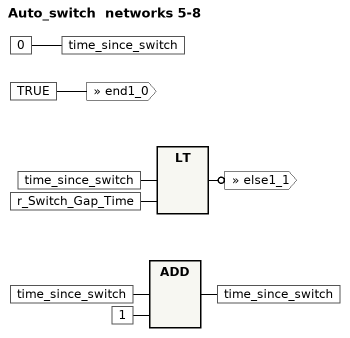
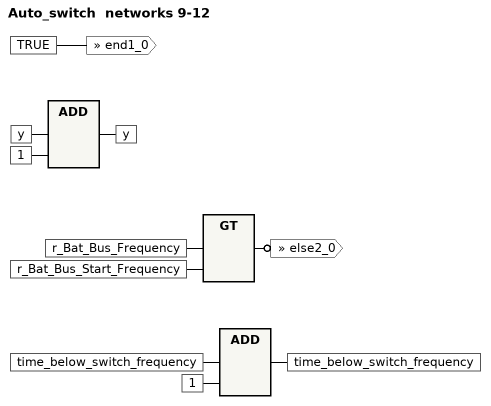
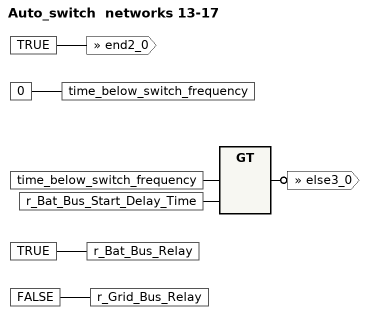
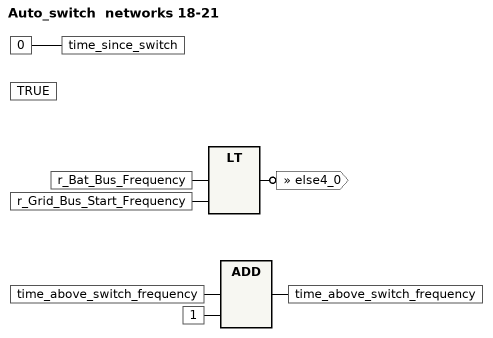
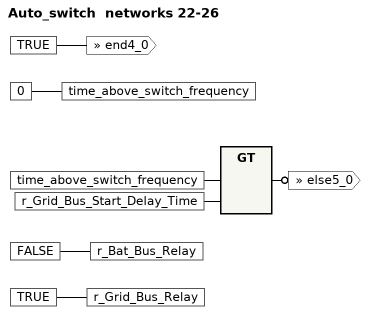
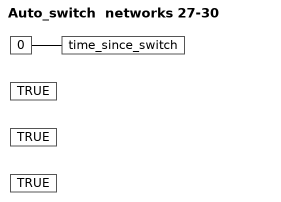
_FBD_ (* Function Block Diagram *)
NETWORK 1 (* this script shuold run every second and / ------ Cases 1 - SAFETY ------ / 1) bat voltage  below 200 	> swtich to gridbus / ------ Cases 2 - NO PENDEL ------ / 2) just switched (wait for r_Switch_Gap_Time) / ------ Cases 3 - LOW FREQUENCY = ENERGY SHORTAGE ------ / 3a) bat frequency below < r_Grid_Bus_Start_Frequency => "reset "to grid counter" / 3b) bat frequency below > r_Grid_Bus_Start_Frequency => "increase "to grid counter" / 3c) "to grid counter" > r_Grid_Bus_Start_Delay_Time => switch of testbus, switch on gridbus relais / ------ Cases 4 - HIGH FREQUENCY = ENERGY SURPLUS ------ / 4a) bat frequency above > r_Bat_Bus_Start_Frequency => "reset "to bat counter" / 4c) "to bat counter" > r_Grid_Bus_Start_Delay_Time => switch of gridbus, switch on testbus relais *)
	ADD(x, 1) => x
NETWORK 2
	NOT LT(r_Bat_Bus_Voltage, 200) => >>else1_0
NETWORK 3 (* case 1 (safety, switching to gridbus) *)
	FALSE => r_Bat_Bus_Relay
NETWORK 4
	TRUE => r_Grid_Bus_Relay
NETWORK 5
	0 => time_since_switch
NETWORK 6
	TRUE => >>end1_0
NETWORK 7 else1_0::
	NOT LT(time_since_switch, r_Switch_Gap_Time) => >>else1_1
NETWORK 8 (* case 2 (already switched recently) *)
	ADD(time_since_switch, 1) => time_since_switch
NETWORK 9
	TRUE => >>end1_0
NETWORK 10 else1_1::
	ADD(y, 1) => y
NETWORK 11 (* CASE 3 / 3a+b *)
	NOT GT(r_Bat_Bus_Frequency, r_Bat_Bus_Start_Frequency) => >>else2_0
NETWORK 12
	ADD(time_below_switch_frequency, 1) => time_below_switch_frequency
NETWORK 13
	TRUE => >>end2_0
NETWORK 14 else2_0::
	0 => time_below_switch_frequency
NETWORK 15 end2_0:: (* 3C time_below_switch_frequency passed >> switching *)
	NOT GT(time_below_switch_frequency, r_Bat_Bus_Start_Delay_Time) => >>else3_0
NETWORK 16
	TRUE => r_Bat_Bus_Relay
NETWORK 17
	FALSE => r_Grid_Bus_Relay
NETWORK 18
	0 => time_since_switch
NETWORK 19 end3_0::
	TRUE
NETWORK 20 else3_0:: (* CASE 4 / 4a+b *)
	NOT LT(r_Bat_Bus_Frequency, r_Grid_Bus_Start_Frequency) => >>else4_0
NETWORK 21
	ADD(time_above_switch_frequency, 1) => time_above_switch_frequency
NETWORK 22
	TRUE => >>end4_0
NETWORK 23 else4_0::
	0 => time_above_switch_frequency
NETWORK 24 end4_0:: (* 4C time_above_switch_frequency passed >> switching *)
	NOT GT(time_above_switch_frequency, r_Grid_Bus_Start_Delay_Time) => >>else5_0
NETWORK 25
	FALSE => r_Bat_Bus_Relay
NETWORK 26
	TRUE => r_Grid_Bus_Relay
NETWORK 27
	0 => time_since_switch
NETWORK 28 end5_0::
	TRUE
NETWORK 29 end1_0::
	TRUE
NETWORK 30 else5_0::
	TRUE
_END_FBD_
END_PROGRAM

(* POU 04. Frequency based Bus Select/Auto_switch_delay, ST *)
PROGRAM Auto_switch_delay
(* ____________________________  USED GLOBAL VARIABLES  ___________________________

VAR_INPUT

	CHP_new_state_grid_bus							:	BOOL; (* request based on frequency *)
	CHP_new_state_battery_bus						:	BOOL; (* request based on frequency *)

	CHP_relay_state_battery_bus   							AT %IX134.1  : BOOL;  (* INVERTED INPUTS *)
	CHP_relay_state_grid_bus   								AT %IX134.2  : BOOL;  (* INVERTED INPUTS *)
	
	CHP_control_internal_contacter_switch_state

END_VAR

VAR_OUTPUT

	Group1_3F_Auto_relay_control_battery_bus							:	BOOL; (* request based on frequency, has delayed switching!! *)
	Group1_3F_Auto_relay_control_battery_bus							:	BOOL; (* request based on frequency, has delayed switching!! *)

END_VAR
*)

VAR
	y: BOOL :=FALSE;
	z: INT;
END_VAR
(* CHP handler uses frequency based switching input to control real CHP swithcing when auto input is high *)
(* CHP handler delays switching, such that the CHP can depower and disconnect before switch *)
(* CHP handler delays on-switching, making sure the CHP is disconnected. *)
(* CHP handler delays on-switching, making sure the CHP will connect to the right bus (in the right mode). *)

(* ____________________________  AUTO SWITCH CONTROL  ___________________________ *)
IF Group1_3F_Selector_auto_bus_select = TRUE THEN
	z := z + 1;
	(*check if wanted state to CHP signal is right, change when required *)
	IF CHP_new_state_grid_bus =TRUE THEN
		CHP_control_Offgrid_request :=FALSE;
		z :=0;
		y := FALSE;
	ELSE
		IF CHP_new_state_battery_bus = TRUE THEN
		CHP_control_Offgrid_request :=TRUE;
		z := 100;
		y := TRUE;
		END_IF;
	END_IF;

	(* perform switch between busses when CHP has disconnceted *)
	IF CHP_control_internal_contacter_switch_state = FALSE THEN

		(* Close bat relais when grid relais is open en bat request is still true*)
		IF CHP_new_state_battery_bus =TRUE  THEN

			IF CHP_relay_state_grid_bus = TRUE THEN (* INVERTED INPUTS *)
				Group1_3F_Auto_relay_control_battery_bus := TRUE;
			END_IF;
			Group1_3F_Auto_relay_control_grid_bus := FALSE; (* Disconnect GRID SCWICH*)
		END_IF;

		(* Close grid relais when bat relais is open en grid request is still true*)
		IF CHP_new_state_grid_bus =TRUE  THEN

			IF CHP_relay_state_battery_bus = TRUE THEN (* INVERTED INPUTS *)
				Group1_3F_Auto_relay_control_grid_bus := TRUE;
			END_IF;
			Group1_3F_Auto_relay_control_battery_bus := FALSE; (* Disconnect *)
		END_IF;
	END_IF;


(* ____________________________  MANUAL CONTROL  ___________________________ *)
ELSE
	z := 200;
	(* check if batbus relais is closed, if so, request offgrid (via wanted state *)
	IF Group1_3F_relay_state_battery_bus = TRUE THEN
		CHP_control_Offgrid_request :=TRUE;
	ELSE (* IF Group1_3F_relay_state_grid_bus THEN *)
		CHP_control_Offgrid_request :=FALSE;
	END_IF;

	Group1_3F_Auto_relay_control_grid_bus := FALSE; (* Disconnect GRID SCWICH*)
	Group1_3F_Auto_relay_control_battery_bus := FALSE; (* Disconnect *)
END_IF;
END_PROGRAM

(* POU 02. Batterybus Frequency to Analog Out/EV_Controller, FBD *)
PROGRAM EV_Controller
VAR
	RAMP_REAL: RAMP_REAL;
	Frequency_to_Analog_Out: Frequency_to_Analog_Out;
	EV_control_control_signal2: INT;
	RAMP_WORD4: RAMP_INT;
END_VAR
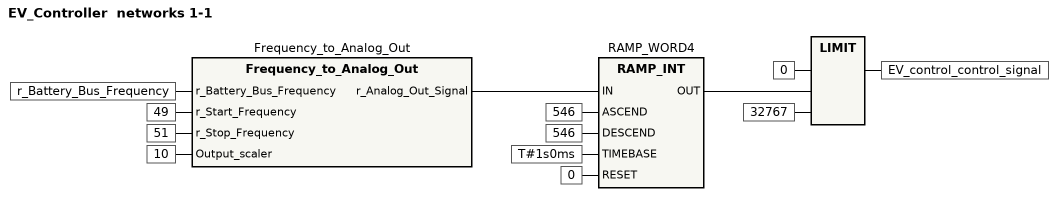
_FBD_ (* Function Block Diagram *)
NETWORK 1
	LIMIT(0, RAMP_WORD4:RAMP_INT(IN: Frequency_to_Analog_Out:Frequency_to_Analog_Out(r_Battery_Bus_Frequency: r_Battery_Bus_Frequency, r_Start_Frequency: 49, r_Stop_Frequency: 51, Output_scaler: 10), ASCEND: 546, DESCEND: 546, TIMEBASE: T#1s0ms, RESET: 0), 32767) => EV_control_control_signal
_END_FBD_
(* the same logic as Structured Text *)
(* Network 1 *)
Frequency_to_Analog_Out(r_Battery_Bus_Frequency := r_Battery_Bus_Frequency, r_Start_Frequency := 49, r_Stop_Frequency := 51, Output_scaler := 10);
RAMP_WORD4(IN := Frequency_to_Analog_Out.r_Analog_Out_Signal, ASCEND := 546, DESCEND := 546, TIMEBASE := T#1s0ms, RESET := 0);
EV_control_control_signal := LIMIT(0, RAMP_WORD4.OUT, 32767);
END_PROGRAM

(* POU 04. Frequency based Bus Select/GroupTest, FBD *)
PROGRAM GroupTest
VAR

	request_grid: BOOL;
	request_testbus: BOOL;
	Delayer: Auto_delayer;
	Switch: Auto_switch_new;
END_VAR
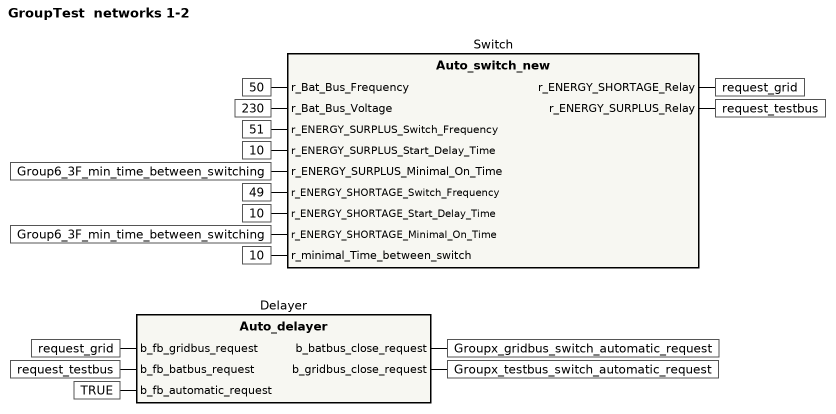
_FBD_ (* Function Block Diagram *)
NETWORK 1
	Switch:Auto_switch_new(r_Bat_Bus_Frequency: 50, r_Bat_Bus_Voltage: 230, r_ENERGY_SURPLUS_Switch_Frequency: 51, r_ENERGY_SURPLUS_Start_Delay_Time: 10, r_ENERGY_SURPLUS_Minimal_On_Time: Group6_3F_min_time_between_switching, r_ENERGY_SHORTAGE_Switch_Frequency: 49, r_ENERGY_SHORTAGE_Start_Delay_Time: 10, r_ENERGY_SHORTAGE_Minimal_On_Time: Group6_3F_min_time_between_switching, r_minimal_Time_between_switch: 10, r_ENERGY_SURPLUS_Relay => request_testbus) => request_grid
NETWORK 2
	Delayer:Auto_delayer(b_fb_gridbus_request: request_grid, b_fb_batbus_request: request_testbus, b_fb_automatic_request: TRUE, b_gridbus_close_request => Groupx_testbus_switch_automatic_request) => Groupx_gridbus_switch_automatic_request
_END_FBD_
(* the same logic as Structured Text *)
(* Network 1 *)
Switch(r_Bat_Bus_Frequency := 50, r_Bat_Bus_Voltage := 230, r_ENERGY_SURPLUS_Switch_Frequency := 51, r_ENERGY_SURPLUS_Start_Delay_Time := 10, r_ENERGY_SURPLUS_Minimal_On_Time := Group6_3F_min_time_between_switching, r_ENERGY_SHORTAGE_Switch_Frequency := 49, r_ENERGY_SHORTAGE_Start_Delay_Time := 10, r_ENERGY_SHORTAGE_Minimal_On_Time := Group6_3F_min_time_between_switching, r_minimal_Time_between_switch := 10);
request_testbus := Switch.r_ENERGY_SURPLUS_Relay;
request_grid := Switch.r_ENERGY_SHORTAGE_Relay;
(* Network 2 *)
Delayer(b_fb_gridbus_request := request_grid, b_fb_batbus_request := request_testbus, b_fb_automatic_request := TRUE);
Groupx_testbus_switch_automatic_request := Delayer.b_gridbus_close_request;
Groupx_gridbus_switch_automatic_request := Delayer.b_batbus_close_request;
END_PROGRAM

(* POU 04. Frequency based Bus Select/init, ST *)
PROGRAM init
VAR

END_VAR
(* frequency based switching is deactivated BY default AND can be activated via modbus *)
IF initialized = FALSE THEN
arSystemState[246] :=Group_control_Frequencybased_bus_selecting_state;  (* default is off *)
arSystemState[247] :=Group_control_min_time_above_switch_frequency;
arSystemState[248] :=Group_control_min_time_below_switch_frequency;
arSystemState[249] :=Group1_3F_Switch_frequency_to_batterybus;
arSystemState[250] :=Group1_3F_Switch_frequency_to_gridbus;
arSystemState[251] :=Group1_3F_min_time_between_switching;
arSystemState[252] :=Group2_3F_Switch_frequency_to_batterybus;
arSystemState[253] :=Group2_3F_Switch_frequency_to_gridbus;
arSystemState[254] :=Group2_3F_min_time_between_switching;
arSystemState[253] :=Group3_3F_Switch_frequency_to_batterybus;
arSystemState[254] :=Group3_3F_Switch_frequency_to_gridbus;
arSystemState[255] :=Group3_3F_min_time_between_switching;
arSystemState[256] :=Group4_3F_Switch_frequency_to_batterybus;
arSystemState[255] :=Group4_3F_Switch_frequency_to_gridbus;
arSystemState[256] :=Group4_3F_min_time_between_switching;
arSystemState[257] :=Group5_3F_Switch_frequency_to_batterybus;
arSystemState[258] :=Group5_3F_Switch_frequency_to_gridbus;
arSystemState[257] :=Group5_3F_min_time_between_switching;
arSystemState[258] :=Group6_3F_Switch_frequency_to_batterybus;
arSystemState[259] :=Group6_3F_Switch_frequency_to_gridbus;
arSystemState[260] :=Group6_3F_min_time_between_switching;
arSystemState[259] :=Group7_3F_Switch_frequency_to_batterybus;
arSystemState[260] :=Group7_3F_Switch_frequency_to_gridbus;
arSystemState[261] :=Group7_3F_min_time_between_switching;
arSystemState[262] :=Group8_3F_Switch_frequency_to_batterybus;
arSystemState[261] :=Group8_3F_Switch_frequency_to_gridbus;
arSystemState[262] :=Group8_3F_min_time_between_switching;
arSystemState[263] :=Group9_3F_Switch_frequency_to_batterybus;
arSystemState[264] :=Group9_3F_Switch_frequency_to_gridbus;
arSystemState[263] :=Group9_3F_min_time_between_switching;
initialized := TRUE;
END_IF;
END_PROGRAM

(* POU Configuration/MODBUS_CONFIGURATION, ST *)
PROGRAM MODBUS_CONFIGURATION
VAR                                
END_VAR                            
(*                                 
   <?xml version="1.0" encoding="UTF-16" standalone="yes"?>
<network xml_structure_version="1" xml_feature_version="1">
	<generator_settings minRTUTaskCycleTimeMs="100" minEthaskCycleTimeMs="5" ethSlaveMultiplier="0.1" rtuInterfaceMultiplier="0.1" taskGeneration="false"/>
	<master_interface type="eth" name="" expanded="true">
		<mb_slave comment="" name="Janitza_UMG5090" expanded="true" type="generic">
			<mb_connection type="eth" transport="UDP" port="502" ip="192.168.1.2" unitid="1" request_delay_ms="0" response_timeout_ms="20"/>
			<generic_vars comment="" expanded="true">
				<generic_var data_type="REAL">
					<generic_params name="PactiveL1" comment="" expanded="false" mb_iotype="unused" mb_access="ro" var_byteorder="B3B4B1B2"/>
					<mb_address explicitAccess="false" FCRead="3" FCWrite="0" ReadMBAddress="2069" WriteMBAddress="0" ReadBitOffset="0" WriteBitOffset="0"/>
				</generic_var>
				<generic_var data_type="REAL">
					<generic_params name="PactiveL2" comment="" expanded="true" mb_iotype="unused" mb_access="ro" var_byteorder="B3B4B1B2"/>
					<mb_address explicitAccess="false" FCRead="3" FCWrite="0" ReadMBAddress="2071" WriteMBAddress="0" ReadBitOffset="0" WriteBitOffset="0"/>
				</generic_var>
				<generic_var data_type="REAL">
					<generic_params name="PactiveL3" comment="" expanded="true" mb_iotype="unused" mb_access="ro" var_byteorder="B3B4B1B2"/>
					<mb_address explicitAccess="false" FCRead="3" FCWrite="0" ReadMBAddress="2073" WriteMBAddress="0" ReadBitOffset="0" WriteBitOffset="0"/>
				</generic_var>
				<generic_var data_type="REAL">
					<generic_params name="PreactiveL1" comment="" expanded="false" mb_iotype="unused" mb_access="ro" var_byteorder="B3B4B1B2"/>
					<mb_address explicitAccess="false" FCRead="3" FCWrite="0" ReadMBAddress="2077" WriteMBAddress="0" ReadBitOffset="0" WriteBitOffset="0"/>
				</generic_var>
				<generic_var data_type="REAL">
					<generic_params name="PreactiveL2" comment="" expanded="true" mb_iotype="unused" mb_access="ro" var_byteorder="B3B4B1B2"/>
					<mb_address explicitAccess="false" FCRead="3" FCWrite="0" ReadMBAddress="2079" WriteMBAddress="0" ReadBitOffset="0" WriteBitOffset="0"/>
				</generic_var>
				<generic_var data_type="REAL">
					<generic_params name="PreactiveL3" comment="" expanded="true" mb_iotype="unused" mb_access="ro" var_byteorder="B3B4B1B2"/>
					<mb_address explicitAccess="false" FCRead="3" FCWrite="0" ReadMBAddress="2081" WriteMBAddress="0" ReadBitOffset="0" WriteBitOffset="0"/>
				</generic_var>
				<generic_var data_type="REAL">
					<generic_params name="VoltageL1" comment="" expanded="true" mb_iotype="unused" mb_access="ro" var_byteorder="B3B4B1B2"/>
					<mb_address explicitAccess="false" FCRead="3" FCWrite="0" ReadMBAddress="2053" WriteMBAddress="0" ReadBitOffset="0" WriteBitOffset="0"/>
				</generic_var>
				<generic_var data_type="REAL">
					<generic_params name="VoltageL2" comment="" expanded="false" mb_iotype="unused" mb_access="ro" var_byteorder="B3B4B1B2"/>
					<mb_address explicitAccess="false" FCRead="3" FCWrite="0" ReadMBAddress="2055" WriteMBAddress="0" ReadBitOffset="0" WriteBitOffset="0"/>
				</generic_var>
				<generic_var data_type="REAL">
					<generic_params name="VoltageL3" comment="" expanded="false" mb_iotype="unused" mb_access="ro" var_byteorder="B3B4B1B2"/>
					<mb_address explicitAccess="false" FCRead="3" FCWrite="0" ReadMBAddress="2057" WriteMBAddress="0" ReadBitOffset="0" WriteBitOffset="0"/>
				</generic_var>
				<generic_var data_type="REAL">
					<generic_params name="VoltageL4" comment="" expanded="false" mb_iotype="unused" mb_access="ro" var_byteorder="B3B4B1B2"/>
					<mb_address explicitAccess="false" FCRead="3" FCWrite="0" ReadMBAddress="2059" WriteMBAddress="0" ReadBitOffset="0" WriteBitOffset="0"/>
				</generic_var>
				<generic_var data_type="REAL">
					<generic_params name="PhaseCurrentL1" comment="" expanded="true" mb_iotype="unused" mb_access="ro" var_byteorder="B3B4B1B2"/>
					<mb_address explicitAccess="false" FCRead="3" FCWrite="0" ReadMBAddress="2061" WriteMBAddress="0" ReadBitOffset="0" WriteBitOffset="0"/>
				</generic_var>
				<generic_var data_type="REAL">
					<generic_params name="PhaseCurrentL2" comment="" expanded="true" mb_iotype="unused" mb_access="ro" var_byteorder="B3B4B1B2"/>
					<mb_address explicitAccess="false" FCRead="3" FCWrite="0" ReadMBAddress="2063" WriteMBAddress="0" ReadBitOffset="0" WriteBitOffset="0"/>
				</generic_var>
				<generic_var data_type="REAL">
					<generic_params name="PhaseCurrentL3" comment="" expanded="true" mb_iotype="unused" mb_access="ro" var_byteorder="B3B4B1B2"/>
					<mb_address explicitAccess="false" FCRead="3" FCWrite="0" ReadMBAddress="2065" WriteMBAddress="0" ReadBitOffset="0" WriteBitOffset="0"/>
				</generic_var>
				<generic_var data_type="REAL">
					<generic_params name="PhaseCurrentLN" comment="" expanded="true" mb_iotype="unused" mb_access="ro" var_byteorder="B3B4B1B2"/>
					<mb_address explicitAccess="false" FCRead="3" FCWrite="0" ReadMBAddress="2067" WriteMBAddress="0" ReadBitOffset="0" WriteBitOffset="0"/>
				</generic_var>
				<generic_var data_type="REAL">
					<generic_params name="FieldRotation" comment="" expanded="true" mb_iotype="unused" mb_access="ro" var_byteorder="B3B4B1B2"/>
					<mb_address explicitAccess="false" FCRead="3" FCWrite="0" ReadMBAddress="2185" WriteMBAddress="0" ReadBitOffset="0" WriteBitOffset="0"/>
				</generic_var>
				<generic_var data_type="REAL">
					<generic_params name="CosPihL1" comment="" expanded="true" mb_iotype="unused" mb_access="ro" var_byteorder="B3B4B1B2"/>
					<mb_address explicitAccess="false" FCRead="3" FCWrite="0" ReadMBAddress="2159" WriteMBAddress="0" ReadBitOffset="0" WriteBitOffset="0"/>
				</generic_var>
				<generic_var data_type="REAL">
					<generic_params name="CosPihL2" comment="" expanded="true" mb_iotype="unused" mb_access="ro" var_byteorder="B3B4B1B2"/>
					<mb_address explicitAccess="false" FCRead="3" FCWrite="0" ReadMBAddress="2161" WriteMBAddress="0" ReadBitOffset="0" WriteBitOffset="0"/>
				</generic_var>
				<generic_var data_type="REAL">
					<generic_params name="CosPihL3" comment="" expanded="true" mb_iotype="unused" mb_access="ro" var_byteorder="B3B4B1B2"/>
					<mb_address explicitAccess="false" FCRead="3" FCWrite="0" ReadMBAddress="2163" WriteMBAddress="0" ReadBitOffset="0" WriteBitOffset="0"/>
				</generic_var>
				<generic_var data_type="REAL">
					<generic_params name="Frequency" comment="" expanded="true" mb_iotype="unused" mb_access="ro" var_byteorder="B3B4B1B2"/>
					<mb_address explicitAccess="false" FCRead="3" FCWrite="0" ReadMBAddress="2175" WriteMBAddress="0" ReadBitOffset="0" WriteBitOffset="0"/>
				</generic_var>
				<generic_var data_type="REAL">
					<generic_params name="PactivetTot" comment="" expanded="false" mb_iotype="unused" mb_access="ro" var_byteorder="B3B4B1B2"/>
					<mb_address explicitAccess="false" FCRead="3" FCWrite="0" ReadMBAddress="2105" WriteMBAddress="0" ReadBitOffset="0" WriteBitOffset="0"/>
				</generic_var>
				<generic_var data_type="REAL">
					<generic_params name="PactivetTotL4" comment="" expanded="false" mb_iotype="unused" mb_access="ro" var_byteorder="B3B4B1B2"/>
					<mb_address explicitAccess="false" FCRead="3" FCWrite="0" ReadMBAddress="2113" WriteMBAddress="0" ReadBitOffset="0" WriteBitOffset="0"/>
				</generic_var>
			</generic_vars>
		</mb_slave>
	</master_interface>
</network>
                              
*)                                 
;                                  
END_PROGRAM

(* POU 02. Batterybus Frequency to Analog Out/other_control_signal, FBD *)
PROGRAM other_control_signal
VAR
	RAMP_REAL: RAMP_REAL;
	Frequency_to_Analog_Out: Frequency_to_Analog_Out;
END_VAR
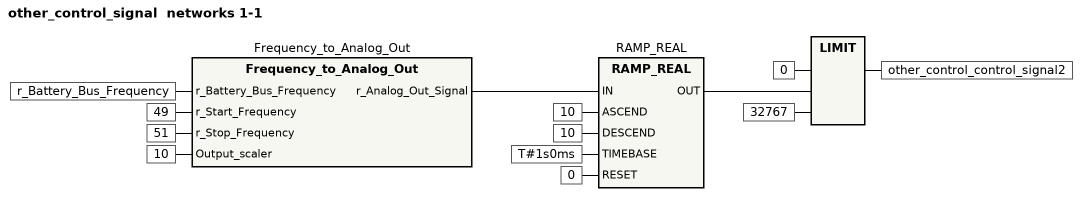
_FBD_ (* Function Block Diagram *)
NETWORK 1
	LIMIT(0, RAMP_REAL:RAMP_REAL(IN: Frequency_to_Analog_Out:Frequency_to_Analog_Out(r_Battery_Bus_Frequency: r_Battery_Bus_Frequency, r_Start_Frequency: 49, r_Stop_Frequency: 51, Output_scaler: 10), ASCEND: 10, DESCEND: 10, TIMEBASE: T#1s0ms, RESET: 0), 32767) => other_control_control_signal2
_END_FBD_
(* the same logic as Structured Text *)
(* Network 1 *)
Frequency_to_Analog_Out(r_Battery_Bus_Frequency := r_Battery_Bus_Frequency, r_Start_Frequency := 49, r_Stop_Frequency := 51, Output_scaler := 10);
RAMP_REAL(IN := Frequency_to_Analog_Out.r_Analog_Out_Signal, ASCEND := 10, DESCEND := 10, TIMEBASE := T#1s0ms, RESET := 0);
other_control_control_signal2 := LIMIT(0, RAMP_REAL.OUT, 32767);
END_PROGRAM

(* POU TheBattery/SOC_real_to_Voltage_Out, ST *)
PROGRAM SOC_real_to_Voltage_Out
VAR

END_VAR
other_control_control_signal := REAL_TO_WORD(6553.6*TheBattery_SOC_real/10);
END_PROGRAM

(* POU 03. Synchroniser Switch control/SynchronizerModbusStateHandler_PRG, ST *)
PROGRAM SynchronizerModbusStateHandler_PRG
VAR

END_VAR
(*___OLD___
IF r_modbus_Synchroniser_state < 1 THEN
		r_modbus_Synchroniser_Denied_Request := TRUE;
		r_modbus_Synchroniser_Close_Request := FALSE;
ELSE
	IF r_modbus_Synchroniser_state > 1.99 THEN
		r_modbus_Synchroniser_Denied_Request := FALSE;
		r_modbus_Synchroniser_Close_Request := TRUE;
	ELSE
		r_modbus_Synchroniser_Denied_Request := FALSE;
		r_modbus_Synchroniser_Close_Request := FALSE;
	END_IF
END_IF
*)
END_PROGRAM

(* POU 04. Frequency based Bus Select/Test, ST *)
PROGRAM Test
VAR

	Test :fbSwitchRelaysBatOrGridBus;
	a: REAL;
	frequencybased_bus_selecting_state: BOOL;
END_VAR
	frequencybased_bus_selecting_state : = arSystemState[999]; (* frequency based switching is deactivated by default and can be activated via modbus *)


Test(
	r_Off_Grid_Bus_Frequency:= r_Battery_Bus_Frequency ,
	r_Off_Grid_Bus_Voltage:= 250,
	r_On_Grid_Start_Frequency:= 49,
	r_On_Grid_Start_Delay_Time:= 2000,
	r_On_Grid_Minimal_On_Time:= 2000 ,
	r_Off_Grid_Start_Frequency:= 51,
	r_Off_Grid_Start_Delay_Time:= 2000,
	r_Switch_Gap_Time:= 2000,
	r_Off_Grid_Minimal_On_Time:= 2000);

(*
	Group1_Switch_frequency_to_batterybus						:  read from mobus;
	Group1_Switch_frequency_to_gridbus							:  REAL 	:= 48;
	Group1_min_time_above_switch frequency						:  INT 		: = 10000; (*ms*)
	Group1_min_time_below_switch frequency						:  INT 		: = 10000; (*ms*)
	Group1_min_time_between_switching							:  INT 		: = 10000; (*ms*)
*)
END_PROGRAM

(* POU 04. Frequency based Bus Select/fbSwitchRelaysBatOrGridBus, SFC *)
FUNCTION_BLOCK fbSwitchRelaysBatOrGridBus
VAR_INPUT

	r_Bat_Bus_Frequency						:	REAL;
	r_Bat_Bus_Voltage							:	REAL;
	r_Grid_Bus_Start_Frequency					:	REAL;
	r_Grid_Bus_Start_Delay_Time				:	REAL;
	r_Grid_Bus_Minimal_On_Time				:	REAL;
	r_Bat_Bus_Start_Frequency					:	REAL;
	r_Bat_Bus_Start_Delay_Time				:	REAL;
	r_Bat_Bus_Minimal_On_Time				:	REAL;
	r_Switch_Gap_Time							: 	REAL;		(* Time between on and off grid relay switching (dead bus gap) *)

END_VAR
VAR_OUTPUT

	r_Grid_Bus_Relay								:	BOOL := TRUE;
	r_Bat_Bus_Relay									:	BOOL;

END_VAR
VAR
	r_Bat_Bus_Min_Voltage 							: 	REAL :=200;
	r_Checked_Grid_Bus_Start_Frequency			:	REAL;
	r_Checked_Bat_Bus_Start_Frequency			:	REAL;

	t_Grid_Bus_Start_Delay_Timer					:	TON;
	t_Bat_Bus_Start_Delay_Timer					:	TON;

END_VAR
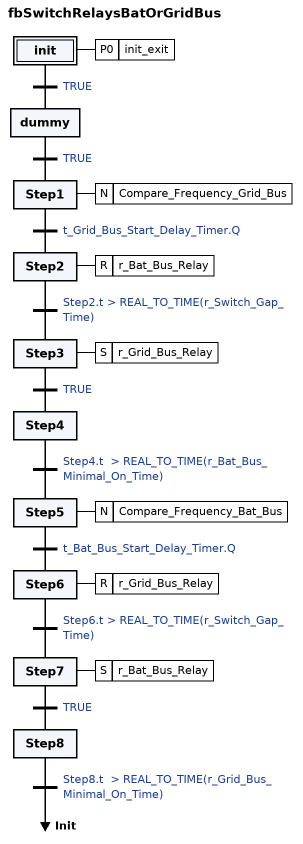
INITIAL_STEP init:
	init_exit(P0);
END_STEP
TRANSITION FROM init TO dummy := TRUE;
END_TRANSITION
STEP dummy:
END_STEP
TRANSITION FROM dummy TO Step1 := TRUE;
END_TRANSITION
STEP Step1:
	Compare_Frequency_Grid_Bus(N);
END_STEP
TRANSITION FROM Step1 TO Step2 := t_Grid_Bus_Start_Delay_Timer.Q;
END_TRANSITION
STEP Step2:
	r_Bat_Bus_Relay(R);
END_STEP
TRANSITION FROM Step2 TO Step3 := Step2.t > REAL_TO_TIME(r_Switch_Gap_Time);
END_TRANSITION
STEP Step3:
	r_Grid_Bus_Relay(S);
END_STEP
TRANSITION FROM Step3 TO Step4 := TRUE;
END_TRANSITION
STEP Step4:
END_STEP
TRANSITION FROM Step4 TO Step5 := Step4.t  > REAL_TO_TIME(r_Bat_Bus_Minimal_On_Time);
END_TRANSITION
STEP Step5:
	Compare_Frequency_Bat_Bus(N);
END_STEP
TRANSITION FROM Step5 TO Step6 := t_Bat_Bus_Start_Delay_Timer.Q;
END_TRANSITION
STEP Step6:
	r_Grid_Bus_Relay(R);
END_STEP
TRANSITION FROM Step6 TO Step7 := Step6.t > REAL_TO_TIME(r_Switch_Gap_Time);
END_TRANSITION
STEP Step7:
	r_Bat_Bus_Relay(S);
END_STEP
TRANSITION FROM Step7 TO Step8 := TRUE;
END_TRANSITION
STEP Step8:
END_STEP
TRANSITION FROM Step8 TO Init := Step8.t  > REAL_TO_TIME(r_Grid_Bus_Minimal_On_Time);
END_TRANSITION

ACTION init_exit:
(* Bat_Bus start frequency should by higher than grid bus start frequency to prevent pendel behaviour of states *)

IF r_Bat_Bus_Start_Frequency > r_Grid_Bus_Start_Frequency THEN

	r_Checked_Bat_Bus_Start_Frequency := r_Bat_Bus_Start_Frequency;
	r_Checked_Grid_Bus_Start_Frequency := r_Grid_Bus_Start_Frequency;

ELSE

	r_Checked_Bat_Bus_Start_Frequency := r_Bat_Bus_Start_Frequency;
	r_Checked_Grid_Bus_Start_Frequency := r_Bat_Bus_Start_Frequency;

END_IF
END_ACTION
END_FUNCTION_BLOCK
ACTION Compare_Frequencies:
(* Bat_Bus start frequency should by higher than grid bus start frequency to prevent pendel behaviour of states *)

IF r_Bat_Bus_Start_Frequency > r_Grid_Bus_Start_Frequency THEN

	r_Checked_Bat_Bus_Start_Frequency := r_Bat_Bus_Start_Frequency;
	r_Checked_Grid_Bus_Start_Frequency := r_Grid_Bus_Start_Frequency;

ELSE

	r_Checked_Bat_Bus_Start_Frequency := r_Bat_Bus_Start_Frequency;
	r_Checked_Grid_Bus_Start_Frequency := r_Bat_Bus_Start_Frequency;

END_IF
END_ACTION
ACTION Compare_Frequency_Bat_Bus:
t_Bat_Bus_Start_Delay_Timer(
	IN:= r_Bat_Bus_Frequency > r_Checked_Bat_Bus_Start_Frequency AND r_Bat_Bus_Voltage > r_Bat_Bus_Min_Voltage,
	PT:= REAL_TO_TIME(r_Bat_Bus_Start_Delay_Time));
END_ACTION
ACTION Compare_Frequency_Grid_Bus:
t_Grid_Bus_Start_Delay_Timer(
	IN:= r_Bat_Bus_Frequency < r_Checked_Grid_Bus_Start_Frequency,
	PT:= REAL_TO_TIME(r_Grid_Bus_Start_Delay_Time));
END_ACTION
ACTION Compare_Frequency_Grid_Bus_old:
t_Grid_Bus_Start_Delay_Timer(
	IN:= r_Bat_Bus_Frequency < r_Checked_Grid_Bus_Start_Frequency,
	PT:= REAL_TO_TIME(r_Grid_Bus_Start_Delay_Time));
END_ACTION
ACTION Compare_Frequency_Grid_Bus_olds:
t_Grid_Bus_Start_Delay_Timer(
	IN:= r_Bat_Bus_Frequency < r_Checked_Grid_Bus_Start_Frequency,
	PT:= REAL_TO_TIME(r_Grid_Bus_Start_Delay_Time));
END_ACTION

(* POU 04. Frequency based Bus Select/test_switch, LD *)
PROGRAM test_switch
VAR
	test: CHP_Switch_Handler;
END_VAR
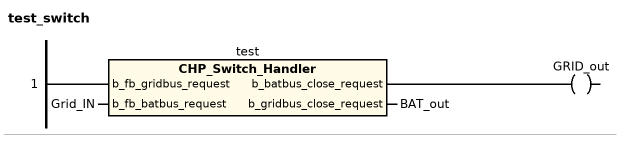
_LD_ (* Ladder Diagram *)
NETWORK 1
	test:CHP_Switch_Handler(b_fb_gridbus_request: *, b_fb_batbus_request: Grid_IN, b_gridbus_close_request => BAT_out) --- (GRID_out)
_END_LD_
(* the same logic as Structured Text *)
(* Network 1 *)
test(b_fb_gridbus_request := TRUE, b_fb_batbus_request := Grid_IN);
BAT_out := test.b_gridbus_close_request;
GRID_out := test.b_batbus_close_request;
END_PROGRAM

(* POU 04. Frequency based Bus Select/CHP_Switch_Handler, ST *)
FUNCTION_BLOCK CHP_Switch_Handler

VAR_INPUT

	b_fb_gridbus_request							:	BOOL; (* request based on frequency, has delayed switching!! *)
	b_fb_batbus_request								:	BOOL; (* request based on frequency, has delayed switching!! *)

END_VAR

VAR_OUTPUT

	b_batbus_close_request							:	BOOL; (* request based on frequency, has delayed switching!! *)
	b_gridbus_close_request							:	BOOL; (* request based on frequency, has delayed switching!! *)

END_VAR

VAR
(* ____________________________  USED GLOBAL VARIABLES  ___________________________ *)
(*
	(* INPUTS *)
	CHP_control_internal_contacter_switch_state  			AT %IX121.15 : BOOL;
	Group1_3F_Selector_auto_bus_select    				AT %IX121.2 : BOOL;
	Group1_3F_relay_state_battery_bus   					AT %IX120.1  : BOOL;
	Group1_3F_relay_state_grid_bus   						AT %IX120.0  : BOOL;

	(* OUTPUTS *)
	Group1_3F_Auto_relay_control_battery_bus   			AT %QX128.1  : BOOL;
	Group1_3F_Auto_relay_control_grid_bus   				AT %QX128.0  : BOOL;
	CHP_control_Offgrid_request    							AT %QX129.4  : BOOL;
*)
	y: BOOL :=FALSE;
	z: INT;
END_VAR
(* CHP handler uses frequency based switching input to control real CHP swithcing when auto input is high *)
(* CHP handler delays switching, such that the CHP can depower and disconnect before switch *)
(* CHP handler delays on-switching, making sure the CHP is disconnected. *)
(* CHP handler delays on-switching, making sure the CHP will connect to the right bus (in the right mode). *)

(* ____________________________  AUTO SWITCH CONTROL  ___________________________ *)
IF Group1_3F_Selector_auto_bus_select = TRUE THEN
	z := z + 1;
	(*check if wanted state to CHP signal is right, change when required *)
	IF b_fb_gridbus_request =TRUE THEN
		CHP_control_Offgrid_request :=FALSE;
		z :=0;
		y := FALSE;
	ELSE
		IF b_fb_batbus_request = TRUE THEN
		CHP_control_Offgrid_request :=TRUE;
		z := 100;
		y := TRUE;
		END_IF;
	END_IF;

	(* perform switch between busses when CHP has disconnceted *)
	IF CHP_control_internal_contacter_switch_state = FALSE THEN

		(* Close bat relais when grid relais is open en bat request is still true*)
		IF b_fb_batbus_request =TRUE  THEN
			b_gridbus_close_request := FALSE; (* Disconnect GRID SCWICH*)
			IF Group1_3F_relay_state_grid_bus = FALSE THEN
				b_batbus_close_request := TRUE;
			END_IF;
		END_IF;

		(* Close grid relais when bat relais is open en grid request is still true*)
		IF b_fb_gridbus_request =TRUE  THEN
			b_batbus_close_request := FALSE; (* Disconnect *)
			IF Group1_3F_relay_state_battery_bus = FALSE THEN
				b_gridbus_close_request := TRUE;
			END_IF;
		END_IF;
	END_IF;


(* ____________________________  MANUAL CONTROL  ___________________________ *)
ELSE
	z := 200;
	(* check if batbus relais is closed, if so, request offgrid (via wanted state *)
	IF Group1_3F_relay_state_battery_bus = TRUE THEN
		CHP_control_Offgrid_request :=TRUE;
	ELSE (* IF Group1_3F_relay_state_grid_bus THEN *)
		CHP_control_Offgrid_request :=FALSE;
	END_IF;
END_IF;
END_FUNCTION_BLOCK

(* POU 08. SD CARD logging/WRITE_CSV/WRITE_DATA, FBD *)
PROGRAM WRITE_DATA
VAR
	FB1				: FbDatalogger;
	xGo				: BOOL		:= TRUE;
	xTrigger			: BOOL;
	Channels			: ARRAY [1.. 80] OF typUserInput;
	Settings			: typConfigDatalogger;
	bDType			: BYTE := 1;
	xFirstCycle			: BOOL := TRUE;
	i: INT;

END_VAR
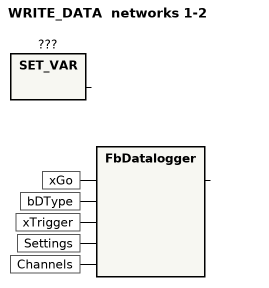
_FBD_ (* Function Block Diagram *)
NETWORK 1
	???:SET_VAR()
NETWORK 2
	FbDatalogger(xGo, bDType, xTrigger, Settings, Channels)
_END_FBD_
(* the same logic as Structured Text *)
(* Network 1: see the listing above *)
(* Network 2 *)
FbDatalogger(xGo, bDType, xTrigger, Settings, Channels);
END_PROGRAM
ACTION SET_VAR:
IF xFirstCycle THEN

	settings.bInterval					:= 3; 						(* 1 = hour, 2= minutes, 3 = seconds *)
	settings.iIntervalFactor			:= 5;						(* number of hours/minutes/seconds, depending on choice b.Interval *)
	settings.sFilename				:= 'Meetdata.csv';				(* Filename csv-file *)
	settings.sPath						:= '/media/sd/';				(* Path where the csv-file is stored *)
	settings.xAppendDate			:= TRUE;					(* When true, the date on the controller is added to the filename*)
	settings.xCyclicLogging			:= TRUE;					(* When true, information is stored cyclic on the controller/SD card *)

	Channels[1].xChannelExists		:= TRUE;
	Channels[1].sChannelName		:= 'PhaseCurrentl2';
	Channels[1].sUnit					:= 'A';
	Channels[1].rAlarmLowerLimit	:= -10000000;
	Channels[1].rAlarmUpperLimit	:= 10000000;

	Channels[2].xChannelExists		:= TRUE;
	Channels[2].sChannelName		:= 'VoltageV31';
	Channels[2].sUnit					:= 'V';
	Channels[2].rAlarmLowerLimit	:= -10000000;
	Channels[2].rAlarmUpperLimit	:= 10000000;

	Channels[3].xChannelExists		:= TRUE;
	Channels[3].sChannelName		:= 'Pactive';
	Channels[3].sUnit					:= 'W';
	Channels[3].rAlarmLowerLimit	:= -10000000;
	Channels[3].rAlarmUpperLimit	:= 10000000;

	Channels[4].xChannelExists		:= TRUE;
	Channels[4].sChannelName		:= 'Preactive';
	Channels[4].sUnit					:= 'VAr';;
	Channels[4].rAlarmLowerLimit	:= -10000000;
	Channels[4].rAlarmUpperLimit	:= 10000000;

	Channels[5].xChannelExists		:= TRUE;
	Channels[5].sChannelName		:= 'ShortCircuitDirectionA';
	Channels[5].sUnit					:= ' ';
	Channels[5].rAlarmLowerLimit	:= -10000000;
	Channels[5].rAlarmUpperLimit	:= 10000000;

	Channels[6].xChannelExists		:= TRUE;
	Channels[6].sChannelName		:= 'ShortCircuitDirectionB';
	Channels[6].sUnit					:= ' ';
	Channels[6].rAlarmLowerLimit	:= -10000000;
	Channels[6].rAlarmUpperLimit	:= 10000000;

	Channels[7].xChannelExists		:= TRUE;
	Channels[7].sChannelName		:= 'Phase1';
	Channels[7].sUnit					:= ' ';
	Channels[7].rAlarmLowerLimit	:= -10000000;
	Channels[7].rAlarmUpperLimit	:= 10000000;

	Channels[8].xChannelExists		:= TRUE;
	Channels[8].sChannelName		:= 'Phase2';
	Channels[8].sUnit					:=  ' ';
	Channels[8].rAlarmLowerLimit	:= -10000000;
	Channels[8].rAlarmUpperLimit	:= 10000000;

	Channels[9].xChannelExists		:= TRUE;
	Channels[9].sChannelName		:= 'Phase3';
	Channels[9].sUnit					:=  ' ';
	Channels[9].rAlarmLowerLimit	:= -10000000;
	Channels[9].rAlarmUpperLimit	:= 10000000;

	Channels[10].xChannelExists		:= TRUE;
	Channels[10].sChannelName		:= 'StatusRemoteSwitching';
	Channels[10].sUnit					:=  ' ';
	Channels[10].rAlarmLowerLimit	:= -10000000;
	Channels[10].rAlarmUpperLimit	:= 10000000;


	Channels[11].xChannelExists		:= TRUE;
	Channels[11].sChannelName		:= 'SwitchLoadBreaker';
	Channels[11].sUnit					:=  ' ';
	Channels[11].rAlarmLowerLimit	:= -10000000;
	Channels[11].rAlarmUpperLimit	:= 10000000;

	Channels[12].xChannelExists		:= TRUE;
	Channels[12].sChannelName		:= 'Bay3CurrentL1';
	Channels[12].sUnit					:=  'A ';
	Channels[12].rAlarmLowerLimit	:= -10000000;
	Channels[12].rAlarmUpperLimit	:= 10000000;

	Channels[13].xChannelExists		:= TRUE;
	Channels[13].sChannelName		:= 'Bay3CurrentL2';
	Channels[13].sUnit					:=  'A ';
	Channels[13].rAlarmLowerLimit	:= -10000000;
	Channels[13].rAlarmUpperLimit	:= 10000000;

	Channels[14].xChannelExists		:= TRUE;
	Channels[14].sChannelName		:= 'Bay3CurrentL3';
	Channels[14].sUnit					:=  'A ';
	Channels[14].rAlarmLowerLimit	:= -10000000;
	Channels[14].rAlarmUpperLimit	:= 10000000;

	Channels[15].xChannelExists		:= TRUE;
	Channels[15].sChannelName		:= 'Bay4CurrentL1';
	Channels[15].sUnit					:=  'A ';
	Channels[15].rAlarmLowerLimit	:= -10000000;
	Channels[15].rAlarmUpperLimit	:= 10000000;

	Channels[16].xChannelExists		:= TRUE;
	Channels[16].sChannelName		:= 'Bay4CurrentL2';
	Channels[16].sUnit					:=  'A ';
	Channels[16].rAlarmLowerLimit	:= -10000000;
	Channels[16].rAlarmUpperLimit	:= 10000000;

	Channels[17].xChannelExists		:= TRUE;
	Channels[17].sChannelName		:= 'Bay4CurrentL3';
	Channels[17].sUnit					:=  'A ';
	Channels[17].rAlarmLowerLimit	:= -10000000;
	Channels[17].rAlarmUpperLimit	:= 10000000;

	xFirstCycle := FALSE;

END_IF

	Channels[1].rValue			:= MBCFG_ModbusSlave.PhaseCurrenL2;
	Channels[2].rValue			:= MBCFG_ModbusSlave.VoltageV31;
	Channels[3].rValue			:= MBCFG_ModbusSlave.Pactive;
	Channels[4].rValue			:= MBCFG_ModbusSlave.Preactive;
	Channels[5].rValue			:= MBCFG_ModbusSlave.ShortCircuitA;
	Channels[6].rValue			:= MBCFG_ModbusSlave.ShortCircuitB;
	Channels[7].rValue			:= MBCFG_ModbusSlave.Phase1;
	Channels[8].rValue			:= MBCFG_ModbusSlave.Phase2;
	Channels[9].rValue			:= MBCFG_ModbusSlave.Phase3;
	Channels[10].rValue			:= MBCFG_ModbusSlave.StatusRemoteSwitching;
	Channels[11].rValue			:= MBCFG_ModbusSlave.SwitchLoadBreaker;
	Channels[12].rValue			:= PQ_1.arCurrent[1];
	Channels[13].rValue			:= PQ_1.arCurrent[2];
	Channels[14].rValue			:= PQ_1.arCurrent[3];
	Channels[15].rValue			:= PQ_2.arCurrent[1];
	Channels[16].rValue			:= PQ_2.arCurrent[2];
	Channels[17].rValue			:= PQ_2.arCurrent[3];





(* For-loop to set the channels to be written on the SD-card *)
END_ACTION

(* POU 08. SD CARD logging/WriteCSVFile, ST *)
PROGRAM WriteCSVFile
(* 	This function block Writes the contents of the data structure to a CSV File

	Required Libraries:
		Standard.lib
		SysLibFile.lib
*)
VAR_INPUT
	sFILENAME 		:STRING(80); (* Filename to store data to (e.g. 'config.csv' 		*)
	typData			:ARRAY [1..iMaxParams] OF typCSV;
	bSeperator		:BYTE :=59;	(* Seperator semicolon:59=;*)
END_VAR
VAR_IN_OUT
	xStart 			:BOOL;	(* Set TRUE to write data, set False to stop.		 *)
END_VAR
VAR_OUTPUT
	sStatus			:STRING;
	iError 			:INT;	(* 00 : Normal Operation	*)
							(* 90 : Can't Open File 	*)
							(* 91 : Can't Close File 	*)
							(* 92 : Can't Write to File 	*)
END_VAR
VAR
	FileOpen		:BOOL := FALSE;
	handle			:DWORD;
	Mode			:STRING[20] := 'rw'; (* read/write *)
	DataString 		:STRING(80);
	i				:INT;
END_VAR
IF xStart THEN
	sStatus := 'Try to open file';
	IF NOT FileOpen THEN
		(* Open File *)
		handle := SysFileOpen(sFileName, Mode);
		IF handle > 0 THEN
			FileOpen := TRUE;
			sStatus := 'File Open OK.';
		ELSE
			iERROR := 90; (* Could not open file. *)
			sStatus := 'Could not open file.';
		END_IF
	END_IF
	
	IF FileOpen THEN
		FOR i := 1 TO iMaxParams DO
				DataString := TypData[i].sDescription;
				DataString := CONCAT(DataString,ASCIIBYTE_TO_STRING(bSeperator));
				DataString := CONCAT(DataString,(TypData[i].Parameter[1]));
	
				DataString := CONCAT(DataString,ASCIIBYTE_TO_STRING(13)); (* CR *)
				DataString := CONCAT(DataString,ASCIIBYTE_TO_STRING(10)); (* LF *)
				(* Write string to file *)
				IF SysFileWrite(handle, ADR(DataString), LEN(DataString)) = 0 THEN
					iERROR := 92; (* Could not write to file *)
					sStatus := 'Could not write file.';
				END_IF
		END_FOR
	END_IF
	
	IF FileOpen THEN
		(* Close file *)
		IF SysFileClose(handle) THEN
			FileOpen := FALSE;
			sStatus := 'File Saved.';
		ELSE
			iERROR := 91; (* Could not close file *)
			sStatus := 'Could not close file.';
		END_IF
		xStart := FALSE;
	END_IF
END_IF
END_PROGRAM

(* POU 06. Mysql Write/Create_Data_Point, ST *)
FUNCTION Create_Data_Point : DataPoint
VAR
		arCurrDataPoint   : DataPoint;
END_VAR
VAR_INPUT

	iSiteCode: INT;
	rTotalApparentPower				: REAL;						(* Total Apparent Power													II Scheinleistung gesamt *)
	rTotalPowerFactorPF				: REAL;						(* Total Power Factor PF 													II Leistungsfaktor_PF gesamt *)

	arFrequency						: ARRAY[1..3] OF REAL;		(* Frequency																II Frequenz *)
	arVoltage_L_N					: ARRAY[1..3] OF REAL;		(* Voltage L-N 																II Spannung Lx N *)
	arCurrent							: ARRAY[1..3] OF REAL;		(* Current 															   		II Strom *)

	(* TODO add the time stamp into buffered items*)

	DCV1 :REAL;
	DCV2 :REAL;

	DCPower1: REAL;
	DCPower2: REAL;

	DCCurr1 : REAL;
	DCCurr2 : REAL;


END_VAR
VAR
END_VAR
	arCurrDataPoint.iSiteCode := iSiteCode;
	arCurrDataPoint.rTotalApparentPower:=rTotalApparentPower;
	arCurrDataPoint.rTotalPowerFactorPF:=rTotalPowerFactorPF;

	arCurrDataPoint.arFrequency_1:=arFrequency[1];
	arCurrDataPoint.arVoltage_L_N_1:=arVoltage_L_N[1];
	arCurrDataPoint.arCurrent_1:=arCurrent[1];
	arCurrDataPoint.arPower_1:=arCurrDataPoint.arCurrent_1*arCurrDataPoint.arVoltage_L_N_1;

	arCurrDataPoint.arFrequency_2:=arFrequency[2];
	arCurrDataPoint.arVoltage_L_N_2:=arVoltage_L_N[2];
	arCurrDataPoint.arCurrent_2:=arCurrent[2];
	arCurrDataPoint.arPower_2:=arCurrDataPoint.arCurrent_2*arCurrDataPoint.arVoltage_L_N_2;


	arCurrDataPoint.arFrequency_3:=arFrequency[3];
	arCurrDataPoint.arVoltage_L_N_3:=arVoltage_L_N[3];
	arCurrDataPoint.arCurrent_3:=arCurrent[3];
	arCurrDataPoint.arPower_3:=arCurrDataPoint.arCurrent_3*arCurrDataPoint.arVoltage_L_N_3;

	arCurrDataPoint.timeStamp := Get_Time();

	arCurrDataPoint.DCV1 := DCV1;
	arCurrDataPoint.DCV2:=DCV2;
	arCurrDataPoint.DCPower1:=DCPower1;
	arCurrDataPoint.DCPower2:=DCPower2;
	arCurrDataPoint.DCCurr2:=DCCurr2;
	arCurrDataPoint.DCCurr2:=DCCurr2;


	Create_Data_Point := arCurrDataPoint;
END_FUNCTION

(* POU 06. Mysql Write/Get_Time, ST *)
FUNCTION Get_Time : REAL
VAR_INPUT

END_VAR
VAR



END_VAR
(* Haal de systeemtijd op *)
Get_Time := DT_TO_REAL(SysRtcGetTime(FALSE));
END_FUNCTION

(* Visualisation power
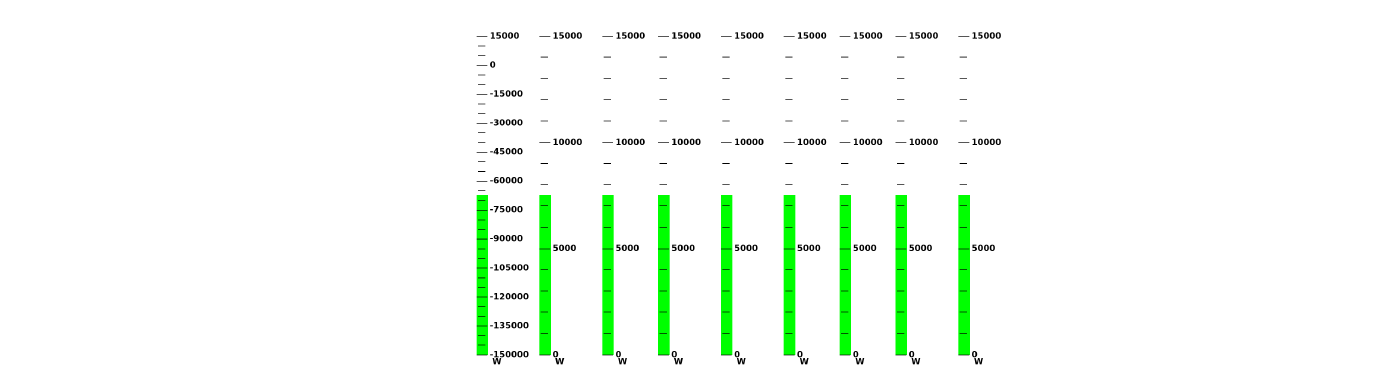
group at (20,60)-(91,571)
  rectangle at (0,0)-(1,1): text "{ExtendedElement},Visu\ElementDLL.ete,1,@Bargraph,71,511,1,1,0,PQ_1.rTotalActivePower,W,%.0f,5000,15000,-150000,15000,0,0,0,0,0,0,0,-13,16,700,Arial,0,255,0,255,0,0,0,0,0,0,0,0,0,,1,0,0,"
  rectangle at (11,248)-(26,463): alarm colour if (PQ_1.rTotalActivePower) < 0; top ((PQ_1.rTotalActivePower * 1.0) - -67500)  * -0.00260606
  rectangle at (27,452)-(66,473): text "-150000"
  rectangle at (27,413)-(66,434): text "-135000"
  rectangle at (27,374)-(66,395): text "-120000"
  rectangle at (27,335)-(66,356): text "-105000"
  rectangle at (27,296)-(66,317): text "-90000"
  rectangle at (27,257)-(66,278): text "-75000"
  rectangle at (27,218)-(66,239): text "-60000"
  rectangle at (27,179)-(66,200): text "-45000"
  rectangle at (27,140)-(66,161): text "-30000"
  rectangle at (27,101)-(66,122): text "-15000"
  rectangle at (27,62)-(66,83): text "0"
  rectangle at (27,23)-(66,44): text "15000"
  rectangle at (25,464)-(51,480): text "W"
group at (110,60)-(181,571)
  rectangle at (0,0)-(1,1): text "{ExtendedElement},Visu\ElementDLL.ete,1,@Bargraph,71,511,1,1,0,PQ_2.rTotalActivePower,W,%.0f,1000,5000,0,15000,0,0,0,0,0,0,0,-13,16,700,Arial,0,255,0,255,0,0,0,0,0,0,0,0,0,,1,0,0,"
  rectangle at (11,248)-(26,463): alarm colour if (PQ_2.rTotalActivePower) < 0; top ((PQ_2.rTotalActivePower * 1.0) - 7500)  * -0.0286667
  rectangle at (27,452)-(66,473): text "0"
  rectangle at (27,309)-(66,330): text "5000"
  rectangle at (27,166)-(66,187): text "10000"
  rectangle at (27,23)-(66,44): text "15000"
  rectangle at (25,464)-(51,480): text "W"
group at (200,60)-(271,571)
  rectangle at (0,0)-(1,1): text "{ExtendedElement},Visu\ElementDLL.ete,1,@Bargraph,71,511,1,1,0,PQ_3.rTotalActivePower,W,%.0f,1000,5000,0,15000,0,0,0,0,0,0,0,-13,16,700,Arial,0,255,0,255,0,0,0,0,0,0,0,0,0,,1,0,0,"
  rectangle at (11,248)-(26,463): alarm colour if (PQ_3.rTotalActivePower) < 0; top ((PQ_3.rTotalActivePower * 1.0) - 7500)  * -0.0286667
  rectangle at (27,452)-(66,473): text "0"
  rectangle at (27,309)-(66,330): text "5000"
  rectangle at (27,166)-(66,187): text "10000"
  rectangle at (27,23)-(66,44): text "15000"
  rectangle at (25,464)-(51,480): text "W"
group at (280,60)-(351,571)
  rectangle at (0,0)-(1,1): text "{ExtendedElement},Visu\ElementDLL.ete,1,@Bargraph,71,511,1,1,0,PQ_4.rTotalActivePower,W,%.0f,1000,5000,0,15000,0,0,0,0,0,0,0,-13,16,700,Arial,0,255,0,255,0,0,0,0,0,0,0,0,0,,1,0,0,"
  rectangle at (11,248)-(26,463): alarm colour if (PQ_4.rTotalActivePower) < 0; top ((PQ_4.rTotalActivePower * 1.0) - 7500)  * -0.0286667
  rectangle at (27,452)-(66,473): text "0"
  rectangle at (27,309)-(66,330): text "5000"
  rectangle at (27,166)-(66,187): text "10000"
  rectangle at (27,23)-(66,44): text "15000"
  rectangle at (25,464)-(51,480): text "W"
group at (370,60)-(441,571)
  rectangle at (0,0)-(1,1): text "{ExtendedElement},Visu\ElementDLL.ete,1,@Bargraph,71,511,1,1,0,PQ_5.rTotalActivePower,W,%.0f,1000,5000,0,15000,0,0,0,0,0,0,0,-13,16,700,Arial,0,255,0,255,0,0,0,0,0,0,0,0,0,,1,0,0,"
  rectangle at (11,248)-(26,463): alarm colour if (PQ_5.rTotalActivePower) < 0; top ((PQ_5.rTotalActivePower * 1.0) - 7500)  * -0.0286667
  rectangle at (27,452)-(66,473): text "0"
  rectangle at (27,309)-(66,330): text "5000"
  rectangle at (27,166)-(66,187): text "10000"
  rectangle at (27,23)-(66,44): text "15000"
  rectangle at (25,464)-(51,480): text "W"
group at (460,60)-(531,571)
  rectangle at (0,0)-(1,1): text "{ExtendedElement},Visu\ElementDLL.ete,1,@Bargraph,71,511,1,1,0,PQ_6.rTotalActivePower,W,%.0f,1000,5000,0,15000,0,0,0,0,0,0,0,-13,16,700,Arial,0,255,0,255,0,0,0,0,0,0,0,0,0,,1,0,0,"
  rectangle at (11,248)-(26,463): alarm colour if (PQ_6.rTotalActivePower) < 0; top ((PQ_6.rTotalActivePower * 1.0) - 7500)  * -0.0286667
  rectangle at (27,452)-(66,473): text "0"
  rectangle at (27,309)-(66,330): text "5000"
  rectangle at (27,166)-(66,187): text "10000"
  rectangle at (27,23)-(66,44): text "15000"
  rectangle at (25,464)-(51,480): text "W"
group at (540,60)-(611,571)
  rectangle at (0,0)-(1,1): text "{ExtendedElement},Visu\ElementDLL.ete,1,@Bargraph,71,511,1,1,0,PQ_7.rTotalActivePower,W,%.0f,1000,5000,0,15000,0,0,0,0,0,0,0,-13,16,700,Arial,0,255,0,255,0,0,0,0,0,0,0,0,0,,1,0,0,"
  rectangle at (11,248)-(26,463): alarm colour if (PQ_7.rTotalActivePower) < 0; top ((PQ_7.rTotalActivePower * 1.0) - 7500)  * -0.0286667
  rectangle at (27,452)-(66,473): text "0"
  rectangle at (27,309)-(66,330): text "5000"
  rectangle at (27,166)-(66,187): text "10000"
  rectangle at (27,23)-(66,44): text "15000"
  rectangle at (25,464)-(51,480): text "W"
group at (620,60)-(691,571)
  rectangle at (0,0)-(1,1): text "{ExtendedElement},Visu\ElementDLL.ete,1,@Bargraph,71,511,1,1,0,PQ_8.rTotalActivePower,W,%.0f,1000,5000,0,15000,0,0,0,0,0,0,0,-13,16,700,Arial,0,255,0,255,0,0,0,0,0,0,0,0,0,,1,0,0,"
  rectangle at (11,248)-(26,463): alarm colour if (PQ_8.rTotalActivePower) < 0; top ((PQ_8.rTotalActivePower * 1.0) - 7500)  * -0.0286667
  rectangle at (27,452)-(66,473): text "0"
  rectangle at (27,309)-(66,330): text "5000"
  rectangle at (27,166)-(66,187): text "10000"
  rectangle at (27,23)-(66,44): text "15000"
  rectangle at (25,464)-(51,480): text "W"
group at (710,60)-(781,571)
  rectangle at (0,0)-(1,1): text "{ExtendedElement},Visu\ElementDLL.ete,1,@Bargraph,71,511,1,1,0,PQ_9.rTotalActivePower,W,%.0f,1000,5000,0,15000,0,0,0,0,0,0,0,-13,16,700,Arial,0,255,0,255,0,0,0,0,0,0,0,0,0,,1,0,0,"
  rectangle at (11,248)-(26,463): alarm colour if (PQ_9.rTotalActivePower) < 0; top ((PQ_9.rTotalActivePower * 1.0) - 7500)  * -0.0286667
  rectangle at (27,452)-(66,473): text "0"
  rectangle at (27,309)-(66,330): text "5000"
  rectangle at (27,166)-(66,187): text "10000"
  rectangle at (27,23)-(66,44): text "15000"
  rectangle at (25,464)-(51,480): text "W"
162 more shapes without text or variables
*)
